// TIA Portal V19 export
VAR_GLOBAL   // PLC tag table "Tag table from XML_1"
END_VAR
